PROGRAM ERROR
VAR
	StopX_a : MC_Stop;
	StopX_b : MC_Stop;
	StopY 	: MC_Stop;
	StopZ 	: MC_Stop;
	
	FB_AXISERRORXa, FB_AXISERRORXb, FB_AXISERRORY, FB_AXISERRORZ : MC_ReadAxisError;
	
	ErrorIDXa 	: DWORD;
	ErrorIDXb 	: DWORD;
	ErrorIDY 	: DWORD;
	ErrorIDZ 	: DWORD;
	
	ErrorAxisXa	: UDINT;
	ErrorAxisXb	: UDINT;
	ErrorAxisY	: UDINT;
	ErrorAxisZ	: UDINT;
END_VAR

//stop all
StopX_a(Axis := gvl.As_Xa,
		Execute := GVL.StopALL);

StopX_b(Axis := gvl.As_Xb,
		Execute := GVL.StopALL);

StopY(Axis := gvl.As_Y,
		Execute := GVL.StopALL);
		
StopZ(Axis := gvl.As_Z,
		Execute := GVL.StopALL);

//error		
FB_AxisErrorXa(Axis := gvl.As_Xa, Enable := TRUE);
FB_AxisErrorXb(Axis := gvl.As_Xb, Enable := TRUE);
FB_AxisErrorY (Axis := gvl.As_Y,  Enable := TRUE);
FB_AxisErrorZ (Axis := gvl.As_Z,  Enable := TRUE);

ErrorIDXa 	:= FB_AxisErrorXa.ErrorID;
ErrorIDXb 	:= FB_AxisErrorXb.ErrorID;
ErrorIDY 	:= FB_AxisErrorY.ErrorID;
ErrorIDZ 	:= FB_AxisErrorZ.ErrorID;

ErrorAxisXa	:= FB_AxisErrorXa.AxisErrorID;
ErrorAxisXb	:= FB_AxisErrorXb.AxisErrorID;
ErrorAxisY	:= FB_AxisErrorY.AxisErrorID;
ErrorAxisZ	:= FB_AxisErrorZ.AxisErrorID;

com.IFerror := FB_axiserrorxa.Error OR FB_axiserrorxb.Error OR FB_axiserrory.Error OR FB_axiserrorz.Error;

END_PROGRAM

(* stored: Version 1.1.0.1, ProductVersion 3.1.4024.2
   POU ERROR: Id {8d68ba2e-431f-4b62-8370-2a49d23c7211}, SpecialFunc None *)
